{attribute addProperty BoxType "EK1122-0000-0018"}
{attribute addProperty Id "Beckhoff_EP2xxxsub_EK1100EK1100_179A0949162A_0001_EP2001_1000_0016EP2001_1F1194F38110.125A_0002_EP2001_1000_0017EP2001_1F1194F38110.125A_0003_EP2001_1000_0018EP2001_1F1194F38110.125A_0004_EP2001_1000_0019EP2001_1F1194F38110.125A_0005_EP2008_0001_0016EP2008_A854BE6D8110.125A_0006_EP2008_0001_0017EP2008_A854BE6D8110.125A_0007_EP2008_0001_0018EP2008_A854BE6D8110.125A_0008_EP2008_0001_0019EP2008_A854BE6D8110.125A_0009_EP2008_0002_0016EP2008_A854BE6D8110.125A_0010_EP2008_0002_0017EP2008_A854BE6D8110.125A_0011_EP2008_0002_0018EP2008_A854BE6D8110.125A_0012_EP2008_0002_0019EP2008_A854BE6D8110.125A_0013_EP2008_0022_0016EP2008_A854BE6D8110.125A_0014_EP2008_0022_0017EP2008_A854BE6D8110.125A_0015_EP2008_0022_0018EP2008_A854BE6D8110.125A_0016_EP2028_0001_0016EP2028_A854BE6D8110.125A_0017_EP2028_0001_0017EP2028_A854BE6D8110.125A_0018_EP2028_0001_0018EP2028_A854BE6D8110.125A_0019_EP2028_0002_0016EP2028_A854BE6D8110.125A_0020_EP2028_0002_0017EP2028_A854BE6D8110.125A_0021_EP2028_0002_0018EP2028_A854BE6D8110.125A_0022_EP2028_0002_0019EP2028_A854BE6D8110.125A_0023_EP2028_0032_0017EP2028_A854BE6D8110.125A_0024_EP2028_0032_0018EP2028_A854BE6D8110.125A_0025_EP2028_0032_0019EP2028_A854BE6D8110.125A_0026_EP2038_0001_0016EP2038_9444C9D314618.25A_0027_EP2038_0001_0017EP2038_9444C9D314618.25A_0028_EP2038_0001_0018EP2038_9444C9D314618.25A_0029_EP2038_0002_0016EP2038_9444C9D314618.25A_0030_EP2038_0002_0017EP2038_9444C9D314618.25A_0031_EP2038_0002_0018EP2038_9444C9D314618.25A_0032_EP2308_0000_0016EP2308_97B4DD118210.25A_0033_EP2308_0000_0017EP2308_97B4DD118210.25A_0034_EP2308_0000_0018EP2308_97B4DD118210.25A_0035_EP2308_0001_0016EP2308_97B4DD118210.25A_0036_EP2308_0001_0017EP2308_97B4DD118210.25A_0037_EP2308_0001_0018EP2308_97B4DD118210.25A_0038_EP2308_0001_0019EP2308_97B4DD118210.25A_0039_EP2308_0002_0016EP2308_97B4DD118210.25A_0040_EP2308_0002_0017EP2308_97B4DD118210.25A_0041_EP2308_0002_0018EP2308_97B4DD118210.25A_0042_EP2308_0002_0019EP2308_97B4DD118210.25A_0043_EP2316_0003_0016EP2316_7CBF98C533842.25A_0044_EP2316_0003_0017EP2316_7CBF98C533842.25A_0045_EP2316_0003_0018EP2316_7CBF98C533842.25A_0046_EP2316_0008_0016EP2316_9E547A1933041.25A_0047_EP2316_0008_0017EP2316_C551FFE833842.25A_0048_EP2316_0008_0018EP2316_4C10EA7633842.25A_0049_EP2316_0008_0019EP2316_7CBF98C533842.25A_0050_EP2316_0008_0020EP2316_7CBF98C533842.25A_0051_EP2316_0008_0021EP2316_7CBF98C533842.25A_0052_EP2318_0001_0016EP2318_97B4DD118210.25A_0053_EP2318_0001_0017EP2318_97B4DD118210.25A_0054_EP2318_0001_0018EP2318_97B4DD118210.25A_0055_EP2318_0001_0019EP2318_97B4DD118210.25A_0056_EP2318_0002_0016EP2318_97B4DD118210.25A_0057_EP2318_0002_0017EP2318_97B4DD118210.25A_0058_EP2318_0002_0018EP2318_97B4DD118210.25A_0059_EP2318_0002_0019EP2318_97B4DD118210.25A_0060_EP2328_0001_0016EP2328_97B4DD118210.25A_0061_EP2328_0001_0017EP2328_97B4DD118210.25A_0062_EP2328_0001_0018EP2328_97B4DD118210.25A_0063_EP2328_0002_0016EP2328_97B4DD118210.25A_0064_EP2328_0002_0017EP2328_97B4DD118210.25A_0065_EP2328_0002_0018EP2328_97B4DD118210.25A_0066_EP2328_0002_0019EP2328_97B4DD118210.25A_0067_EP2328_1061_0016EP2328_FBC9733E8210.25A_0068_EP2338_0001_0016EP2338_F9A026BF14618.25A_0069_EP2338_0001_0017EP2338_F9A026BF14618.25A_0070_EP2338_0001_0018EP2338_538B459D14618.25A_0071_EP2338_0001_0019EP2338_538B459D14618.25A_0072_EP2338_0001_0020EP2338_538B459D14618.25A_0073_EP2338_0001_0021EP2338_538B459D14618.25A_0074_EP2338_0001_0022EP2338_538B459D14618.25A_0075_EP2338_0001_0023EP2338_538B459D14618.25A_0076_EP2338_0002_0016EP2338_F9A026BF14618.25A_0077_EP2338_0002_0017EP2338_F9A026BF14618.25A_0078_EP2338_0002_0018EP2338_538B459D14618.25A_0079_EP2338_0002_0019EP2338_538B459D14618.25A_0080_EP2338_0002_0020EP2338_538B459D14618.25A_0081_EP2338_0002_0021EP2338_538B459D14618.25A_0082_EP2338_0002_0022EP2338_538B459D14618.25A_0083_EP2338_0002_0023EP2338_538B459D14618.25A_0084_EP2338_1001_0016EP2338_538B459D14618.25A_0085_EP2338_1001_0017EP2338_538B459D14618.25A_0086_EP2338_1001_0018EP2338_538B459D14618.25A_0087_EP2338_1002_0016EP2338_538B459D14618.25A_0088_EP2338_1002_0017EP2338_538B459D14618.25A_0089_EP2338_1002_0018EP2338_538B459D14618.25A_0090_EP2339_0003_0016EP2339_41D05C2438648.25A_0092_EP2339_0021_0016EP2339_FC6D243732240.25A_0093_EP2339_0021_0017EP2339_BBE0865932240.25A_0094_EP2339_0021_0018EP2339_BBE0865932240.25A_0095_EP2339_0021_0019EP2339_9219B49827434.25A_0096_EP2339_0021_0020EP2339_9219B49827434.25A_0097_EP2339_0022_0016EP2339_D59416F627434.25A_0098_EP2339_0022_0017EP2339_9219B49827434.25A_0099_EP2339_0022_0018EP2339_9219B49827434.25A_0100_EP2339_0022_0019EP2339_9219B49827434.25A_0101_EP2339_0042_0017EP2339_F4D25F8A8234359738378.25A_0102_EP2339_0042_0018EP2339_90CE4E13429496718668719476722.25A_0103_EP2339_0121_0016EP2339_9219B49827434.25A_0104_EP2349_0021_0016EP2349_9219B49827434.25A_0105_EP2349_0021_0017EP2349_9219B49827434.25A_0106_EP2349_0021_0018EP2349_9219B49827434.25A_0107_EP2349_0022_0016EP2349_9219B49827434.25A_0108_EP2349_0022_0017EP2349_9219B49827434.25A_0109_EP2349_0022_0018EP2349_9219B49827434.25A_0110_EP2624_0002_0016EP2624_4E3C7537496.125A_0111_EP2624_0002_0017EP2624_4E3C7537496.125A_0112_EP2624_0002_0018EP2624_4E3C7537496.125A_0113_EP2624_0002_0019EP2624_4E3C7537496.125A_0114_EP2809_0021_0016EP2809_859F43D214518.125A_0115_EP2809_0021_0017EP2809_859F43D214518.125A_0116_EP2809_0021_0018EP2809_859F43D214518.125A_0117_EP2809_0022_0016EP2809_859F43D214518.125A_0118_EP2809_0022_0017EP2809_859F43D214518.125A_0119_EP2809_0022_0018EP2809_859F43D214518.125A_0120_EP2809_0042_0017EP2809_15BF513E429496724934359738362.125A_0121_EP2809_0042_0018EP2809_556C4F60429496724934359738362.125A_0122_EP2816_0003_0016EP2816_E74B64DB39449.25A_0123_EP2816_0004_0016EP2816_68098FB020926.125A_0124_EP2816_0004_0017EP2816_E74B64DB39449.25A_0125_EP2816_0004_0018EP2816_E74B64DB39449.25A_0126_EP2816_0008_0016EP2816_18670F0939449.25A_0127_EP2816_0008_0017EP2816_18670F0939449.25A_0128_EP2816_0008_0018EP2816_5EA583C239449.25A_0129_EP2816_0008_0019EP2816_907EDA0F39449.25A_0130_EP2816_0008_0020EP2816_907EDA0F39449.25A_0131_EP2816_0008_0021EP2816_907EDA0F39449.25A_0132_EP2816_0010_0016EP2816_18670F0939449.25A_0133_EP2816_0010_0017EP2816_18670F0939449.25A_0134_EP2816_0010_0018EP2816_5EA583C239449.25A_0135_EP2816_0010_0019EP2816_907EDA0F39449.25A_0136_EP2816_0010_0020EP2816_907EDA0F39449.25A_0137_EP2816_0010_0021EP2816_907EDA0F39449.25A_0138_EP2817_0008_0016EP2817_AE3316D954668.25A_0139_EP2817_0008_0017EP2817_AE3316D954668.25A_0140_EP2817_0008_0018EP2817_AE3316D954668.25A_0141_EP2817_0008_0019EP2817_AE3316D954668.25"}
{attribute addProperty CRC "3477339297"}
{attribute addProperty SizeInBites "25538"}
{attribute addProperty SizeInBytes "171798695032.25"}
TYPE Beckhoff_EP2xxxEK1122_CF43FCA1 EXTENDS EK1122_179A0949 :
STRUCT
	{attribute addProperty Name "Beckhoff_EP2xxxsub_EK1100"}
	Beckhoff_EP2xxxsub_EK1100 : EK1100_179A0949;
	{attribute addProperty Name "A_0001_EP2001_1000_0016"}
	A_0001_EP2001_1000_0016 : EP2001_1F1194F3;
	{attribute addProperty Name "A_0002_EP2001_1000_0017"}
	A_0002_EP2001_1000_0017 : EP2001_1F1194F3;
	{attribute addProperty Name "A_0003_EP2001_1000_0018"}
	A_0003_EP2001_1000_0018 : EP2001_1F1194F3;
	{attribute addProperty Name "A_0004_EP2001_1000_0019"}
	A_0004_EP2001_1000_0019 : EP2001_1F1194F3;
	{attribute addProperty Name "A_0005_EP2008_0001_0016"}
	A_0005_EP2008_0001_0016 : EP2008_A854BE6D;
	{attribute addProperty Name "A_0006_EP2008_0001_0017"}
	A_0006_EP2008_0001_0017 : EP2008_A854BE6D;
	{attribute addProperty Name "A_0007_EP2008_0001_0018"}
	A_0007_EP2008_0001_0018 : EP2008_A854BE6D;
	{attribute addProperty Name "A_0008_EP2008_0001_0019"}
	A_0008_EP2008_0001_0019 : EP2008_A854BE6D;
	{attribute addProperty Name "A_0009_EP2008_0002_0016"}
	A_0009_EP2008_0002_0016 : EP2008_A854BE6D;
	{attribute addProperty Name "A_0010_EP2008_0002_0017"}
	A_0010_EP2008_0002_0017 : EP2008_A854BE6D;
	{attribute addProperty Name "A_0011_EP2008_0002_0018"}
	A_0011_EP2008_0002_0018 : EP2008_A854BE6D;
	{attribute addProperty Name "A_0012_EP2008_0002_0019"}
	A_0012_EP2008_0002_0019 : EP2008_A854BE6D;
	{attribute addProperty Name "A_0013_EP2008_0022_0016"}
	A_0013_EP2008_0022_0016 : EP2008_A854BE6D;
	{attribute addProperty Name "A_0014_EP2008_0022_0017"}
	A_0014_EP2008_0022_0017 : EP2008_A854BE6D;
	{attribute addProperty Name "A_0015_EP2008_0022_0018"}
	A_0015_EP2008_0022_0018 : EP2008_A854BE6D;
	{attribute addProperty Name "A_0016_EP2028_0001_0016"}
	A_0016_EP2028_0001_0016 : EP2028_A854BE6D;
	{attribute addProperty Name "A_0017_EP2028_0001_0017"}
	A_0017_EP2028_0001_0017 : EP2028_A854BE6D;
	{attribute addProperty Name "A_0018_EP2028_0001_0018"}
	A_0018_EP2028_0001_0018 : EP2028_A854BE6D;
	{attribute addProperty Name "A_0019_EP2028_0002_0016"}
	A_0019_EP2028_0002_0016 : EP2028_A854BE6D;
	{attribute addProperty Name "A_0020_EP2028_0002_0017"}
	A_0020_EP2028_0002_0017 : EP2028_A854BE6D;
	{attribute addProperty Name "A_0021_EP2028_0002_0018"}
	A_0021_EP2028_0002_0018 : EP2028_A854BE6D;
	{attribute addProperty Name "A_0022_EP2028_0002_0019"}
	A_0022_EP2028_0002_0019 : EP2028_A854BE6D;
	{attribute addProperty Name "A_0023_EP2028_0032_0017"}
	A_0023_EP2028_0032_0017 : EP2028_A854BE6D;
	{attribute addProperty Name "A_0024_EP2028_0032_0018"}
	A_0024_EP2028_0032_0018 : EP2028_A854BE6D;
	{attribute addProperty Name "A_0025_EP2028_0032_0019"}
	A_0025_EP2028_0032_0019 : EP2028_A854BE6D;
	{attribute addProperty Name "A_0026_EP2038_0001_0016"}
	A_0026_EP2038_0001_0016 : EP2038_9444C9D3;
	{attribute addProperty Name "A_0027_EP2038_0001_0017"}
	A_0027_EP2038_0001_0017 : EP2038_9444C9D3;
	{attribute addProperty Name "A_0028_EP2038_0001_0018"}
	A_0028_EP2038_0001_0018 : EP2038_9444C9D3;
	{attribute addProperty Name "A_0029_EP2038_0002_0016"}
	A_0029_EP2038_0002_0016 : EP2038_9444C9D3;
	{attribute addProperty Name "A_0030_EP2038_0002_0017"}
	A_0030_EP2038_0002_0017 : EP2038_9444C9D3;
	{attribute addProperty Name "A_0031_EP2038_0002_0018"}
	A_0031_EP2038_0002_0018 : EP2038_9444C9D3;
	{attribute addProperty Name "A_0032_EP2308_0000_0016"}
	A_0032_EP2308_0000_0016 : EP2308_97B4DD11;
	{attribute addProperty Name "A_0033_EP2308_0000_0017"}
	A_0033_EP2308_0000_0017 : EP2308_97B4DD11;
	{attribute addProperty Name "A_0034_EP2308_0000_0018"}
	A_0034_EP2308_0000_0018 : EP2308_97B4DD11;
	{attribute addProperty Name "A_0035_EP2308_0001_0016"}
	A_0035_EP2308_0001_0016 : EP2308_97B4DD11;
	{attribute addProperty Name "A_0036_EP2308_0001_0017"}
	A_0036_EP2308_0001_0017 : EP2308_97B4DD11;
	{attribute addProperty Name "A_0037_EP2308_0001_0018"}
	A_0037_EP2308_0001_0018 : EP2308_97B4DD11;
	{attribute addProperty Name "A_0038_EP2308_0001_0019"}
	A_0038_EP2308_0001_0019 : EP2308_97B4DD11;
	{attribute addProperty Name "A_0039_EP2308_0002_0016"}
	A_0039_EP2308_0002_0016 : EP2308_97B4DD11;
	{attribute addProperty Name "A_0040_EP2308_0002_0017"}
	A_0040_EP2308_0002_0017 : EP2308_97B4DD11;
	{attribute addProperty Name "A_0041_EP2308_0002_0018"}
	A_0041_EP2308_0002_0018 : EP2308_97B4DD11;
	{attribute addProperty Name "A_0042_EP2308_0002_0019"}
	A_0042_EP2308_0002_0019 : EP2308_97B4DD11;
	{attribute addProperty Name "A_0043_EP2316_0003_0016"}
	A_0043_EP2316_0003_0016 : EP2316_7CBF98C5;
	{attribute addProperty Name "A_0044_EP2316_0003_0017"}
	A_0044_EP2316_0003_0017 : EP2316_7CBF98C5;
	{attribute addProperty Name "A_0045_EP2316_0003_0018"}
	A_0045_EP2316_0003_0018 : EP2316_7CBF98C5;
	{attribute addProperty Name "A_0046_EP2316_0008_0016"}
	A_0046_EP2316_0008_0016 : EP2316_9E547A19;
	{attribute addProperty Name "A_0047_EP2316_0008_0017"}
	A_0047_EP2316_0008_0017 : EP2316_C551FFE8;
	{attribute addProperty Name "A_0048_EP2316_0008_0018"}
	A_0048_EP2316_0008_0018 : EP2316_4C10EA76;
	{attribute addProperty Name "A_0049_EP2316_0008_0019"}
	A_0049_EP2316_0008_0019 : EP2316_7CBF98C5;
	{attribute addProperty Name "A_0050_EP2316_0008_0020"}
	A_0050_EP2316_0008_0020 : EP2316_7CBF98C5;
	{attribute addProperty Name "A_0051_EP2316_0008_0021"}
	A_0051_EP2316_0008_0021 : EP2316_7CBF98C5;
	{attribute addProperty Name "A_0052_EP2318_0001_0016"}
	A_0052_EP2318_0001_0016 : EP2318_97B4DD11;
	{attribute addProperty Name "A_0053_EP2318_0001_0017"}
	A_0053_EP2318_0001_0017 : EP2318_97B4DD11;
	{attribute addProperty Name "A_0054_EP2318_0001_0018"}
	A_0054_EP2318_0001_0018 : EP2318_97B4DD11;
	{attribute addProperty Name "A_0055_EP2318_0001_0019"}
	A_0055_EP2318_0001_0019 : EP2318_97B4DD11;
	{attribute addProperty Name "A_0056_EP2318_0002_0016"}
	A_0056_EP2318_0002_0016 : EP2318_97B4DD11;
	{attribute addProperty Name "A_0057_EP2318_0002_0017"}
	A_0057_EP2318_0002_0017 : EP2318_97B4DD11;
	{attribute addProperty Name "A_0058_EP2318_0002_0018"}
	A_0058_EP2318_0002_0018 : EP2318_97B4DD11;
	{attribute addProperty Name "A_0059_EP2318_0002_0019"}
	A_0059_EP2318_0002_0019 : EP2318_97B4DD11;
	{attribute addProperty Name "A_0060_EP2328_0001_0016"}
	A_0060_EP2328_0001_0016 : EP2328_97B4DD11;
	{attribute addProperty Name "A_0061_EP2328_0001_0017"}
	A_0061_EP2328_0001_0017 : EP2328_97B4DD11;
	{attribute addProperty Name "A_0062_EP2328_0001_0018"}
	A_0062_EP2328_0001_0018 : EP2328_97B4DD11;
	{attribute addProperty Name "A_0063_EP2328_0002_0016"}
	A_0063_EP2328_0002_0016 : EP2328_97B4DD11;
	{attribute addProperty Name "A_0064_EP2328_0002_0017"}
	A_0064_EP2328_0002_0017 : EP2328_97B4DD11;
	{attribute addProperty Name "A_0065_EP2328_0002_0018"}
	A_0065_EP2328_0002_0018 : EP2328_97B4DD11;
	{attribute addProperty Name "A_0066_EP2328_0002_0019"}
	A_0066_EP2328_0002_0019 : EP2328_97B4DD11;
	{attribute addProperty Name "A_0067_EP2328_1061_0016"}
	A_0067_EP2328_1061_0016 : EP2328_FBC9733E;
	{attribute addProperty Name "A_0068_EP2338_0001_0016"}
	A_0068_EP2338_0001_0016 : EP2338_F9A026BF;
	{attribute addProperty Name "A_0069_EP2338_0001_0017"}
	A_0069_EP2338_0001_0017 : EP2338_F9A026BF;
	{attribute addProperty Name "A_0070_EP2338_0001_0018"}
	A_0070_EP2338_0001_0018 : EP2338_538B459D;
	{attribute addProperty Name "A_0071_EP2338_0001_0019"}
	A_0071_EP2338_0001_0019 : EP2338_538B459D;
	{attribute addProperty Name "A_0072_EP2338_0001_0020"}
	A_0072_EP2338_0001_0020 : EP2338_538B459D;
	{attribute addProperty Name "A_0073_EP2338_0001_0021"}
	A_0073_EP2338_0001_0021 : EP2338_538B459D;
	{attribute addProperty Name "A_0074_EP2338_0001_0022"}
	A_0074_EP2338_0001_0022 : EP2338_538B459D;
	{attribute addProperty Name "A_0075_EP2338_0001_0023"}
	A_0075_EP2338_0001_0023 : EP2338_538B459D;
	{attribute addProperty Name "A_0076_EP2338_0002_0016"}
	A_0076_EP2338_0002_0016 : EP2338_F9A026BF;
	{attribute addProperty Name "A_0077_EP2338_0002_0017"}
	A_0077_EP2338_0002_0017 : EP2338_F9A026BF;
	{attribute addProperty Name "A_0078_EP2338_0002_0018"}
	A_0078_EP2338_0002_0018 : EP2338_538B459D;
	{attribute addProperty Name "A_0079_EP2338_0002_0019"}
	A_0079_EP2338_0002_0019 : EP2338_538B459D;
	{attribute addProperty Name "A_0080_EP2338_0002_0020"}
	A_0080_EP2338_0002_0020 : EP2338_538B459D;
	{attribute addProperty Name "A_0081_EP2338_0002_0021"}
	A_0081_EP2338_0002_0021 : EP2338_538B459D;
	{attribute addProperty Name "A_0082_EP2338_0002_0022"}
	A_0082_EP2338_0002_0022 : EP2338_538B459D;
	{attribute addProperty Name "A_0083_EP2338_0002_0023"}
	A_0083_EP2338_0002_0023 : EP2338_538B459D;
	{attribute addProperty Name "A_0084_EP2338_1001_0016"}
	A_0084_EP2338_1001_0016 : EP2338_538B459D;
	{attribute addProperty Name "A_0085_EP2338_1001_0017"}
	A_0085_EP2338_1001_0017 : EP2338_538B459D;
	{attribute addProperty Name "A_0086_EP2338_1001_0018"}
	A_0086_EP2338_1001_0018 : EP2338_538B459D;
	{attribute addProperty Name "A_0087_EP2338_1002_0016"}
	A_0087_EP2338_1002_0016 : EP2338_538B459D;
	{attribute addProperty Name "A_0088_EP2338_1002_0017"}
	A_0088_EP2338_1002_0017 : EP2338_538B459D;
	{attribute addProperty Name "A_0089_EP2338_1002_0018"}
	A_0089_EP2338_1002_0018 : EP2338_538B459D;
	{attribute addProperty Name "A_0090_EP2339_0003_0016"}
	A_0090_EP2339_0003_0016 : EP2339_41D05C24;
	{attribute addProperty Name "A_0092_EP2339_0021_0016"}
	A_0092_EP2339_0021_0016 : EP2339_FC6D2437;
	{attribute addProperty Name "A_0093_EP2339_0021_0017"}
	A_0093_EP2339_0021_0017 : EP2339_BBE08659;
	{attribute addProperty Name "A_0094_EP2339_0021_0018"}
	A_0094_EP2339_0021_0018 : EP2339_BBE08659;
	{attribute addProperty Name "A_0095_EP2339_0021_0019"}
	A_0095_EP2339_0021_0019 : EP2339_9219B498;
	{attribute addProperty Name "A_0096_EP2339_0021_0020"}
	A_0096_EP2339_0021_0020 : EP2339_9219B498;
	{attribute addProperty Name "A_0097_EP2339_0022_0016"}
	A_0097_EP2339_0022_0016 : EP2339_D59416F6;
	{attribute addProperty Name "A_0098_EP2339_0022_0017"}
	A_0098_EP2339_0022_0017 : EP2339_9219B498;
	{attribute addProperty Name "A_0099_EP2339_0022_0018"}
	A_0099_EP2339_0022_0018 : EP2339_9219B498;
	{attribute addProperty Name "A_0100_EP2339_0022_0019"}
	A_0100_EP2339_0022_0019 : EP2339_9219B498;
	{attribute addProperty Name "A_0101_EP2339_0042_0017"}
	A_0101_EP2339_0042_0017 : EP2339_F4D25F8A;
	{attribute addProperty Name "A_0102_EP2339_0042_0018"}
	A_0102_EP2339_0042_0018 : EP2339_90CE4E13;
	{attribute addProperty Name "A_0103_EP2339_0121_0016"}
	A_0103_EP2339_0121_0016 : EP2339_9219B498;
	{attribute addProperty Name "A_0104_EP2349_0021_0016"}
	A_0104_EP2349_0021_0016 : EP2349_9219B498;
	{attribute addProperty Name "A_0105_EP2349_0021_0017"}
	A_0105_EP2349_0021_0017 : EP2349_9219B498;
	{attribute addProperty Name "A_0106_EP2349_0021_0018"}
	A_0106_EP2349_0021_0018 : EP2349_9219B498;
	{attribute addProperty Name "A_0107_EP2349_0022_0016"}
	A_0107_EP2349_0022_0016 : EP2349_9219B498;
	{attribute addProperty Name "A_0108_EP2349_0022_0017"}
	A_0108_EP2349_0022_0017 : EP2349_9219B498;
	{attribute addProperty Name "A_0109_EP2349_0022_0018"}
	A_0109_EP2349_0022_0018 : EP2349_9219B498;
	{attribute addProperty Name "A_0110_EP2624_0002_0016"}
	A_0110_EP2624_0002_0016 : EP2624_4E3C7537;
	{attribute addProperty Name "A_0111_EP2624_0002_0017"}
	A_0111_EP2624_0002_0017 : EP2624_4E3C7537;
	{attribute addProperty Name "A_0112_EP2624_0002_0018"}
	A_0112_EP2624_0002_0018 : EP2624_4E3C7537;
	{attribute addProperty Name "A_0113_EP2624_0002_0019"}
	A_0113_EP2624_0002_0019 : EP2624_4E3C7537;
	{attribute addProperty Name "A_0114_EP2809_0021_0016"}
	A_0114_EP2809_0021_0016 : EP2809_859F43D2;
	{attribute addProperty Name "A_0115_EP2809_0021_0017"}
	A_0115_EP2809_0021_0017 : EP2809_859F43D2;
	{attribute addProperty Name "A_0116_EP2809_0021_0018"}
	A_0116_EP2809_0021_0018 : EP2809_859F43D2;
	{attribute addProperty Name "A_0117_EP2809_0022_0016"}
	A_0117_EP2809_0022_0016 : EP2809_859F43D2;
	{attribute addProperty Name "A_0118_EP2809_0022_0017"}
	A_0118_EP2809_0022_0017 : EP2809_859F43D2;
	{attribute addProperty Name "A_0119_EP2809_0022_0018"}
	A_0119_EP2809_0022_0018 : EP2809_859F43D2;
	{attribute addProperty Name "A_0120_EP2809_0042_0017"}
	A_0120_EP2809_0042_0017 : EP2809_15BF513E;
	{attribute addProperty Name "A_0121_EP2809_0042_0018"}
	A_0121_EP2809_0042_0018 : EP2809_556C4F60;
	{attribute addProperty Name "A_0122_EP2816_0003_0016"}
	A_0122_EP2816_0003_0016 : EP2816_E74B64DB;
	{attribute addProperty Name "A_0123_EP2816_0004_0016"}
	A_0123_EP2816_0004_0016 : EP2816_68098FB0;
	{attribute addProperty Name "A_0124_EP2816_0004_0017"}
	A_0124_EP2816_0004_0017 : EP2816_E74B64DB;
	{attribute addProperty Name "A_0125_EP2816_0004_0018"}
	A_0125_EP2816_0004_0018 : EP2816_E74B64DB;
	{attribute addProperty Name "A_0126_EP2816_0008_0016"}
	A_0126_EP2816_0008_0016 : EP2816_18670F09;
	{attribute addProperty Name "A_0127_EP2816_0008_0017"}
	A_0127_EP2816_0008_0017 : EP2816_18670F09;
	{attribute addProperty Name "A_0128_EP2816_0008_0018"}
	A_0128_EP2816_0008_0018 : EP2816_5EA583C2;
	{attribute addProperty Name "A_0129_EP2816_0008_0019"}
	A_0129_EP2816_0008_0019 : EP2816_907EDA0F;
	{attribute addProperty Name "A_0130_EP2816_0008_0020"}
	A_0130_EP2816_0008_0020 : EP2816_907EDA0F;
	{attribute addProperty Name "A_0131_EP2816_0008_0021"}
	A_0131_EP2816_0008_0021 : EP2816_907EDA0F;
	{attribute addProperty Name "A_0132_EP2816_0010_0016"}
	A_0132_EP2816_0010_0016 : EP2816_18670F09;
	{attribute addProperty Name "A_0133_EP2816_0010_0017"}
	A_0133_EP2816_0010_0017 : EP2816_18670F09;
	{attribute addProperty Name "A_0134_EP2816_0010_0018"}
	A_0134_EP2816_0010_0018 : EP2816_5EA583C2;
	{attribute addProperty Name "A_0135_EP2816_0010_0019"}
	A_0135_EP2816_0010_0019 : EP2816_907EDA0F;
	{attribute addProperty Name "A_0136_EP2816_0010_0020"}
	A_0136_EP2816_0010_0020 : EP2816_907EDA0F;
	{attribute addProperty Name "A_0137_EP2816_0010_0021"}
	A_0137_EP2816_0010_0021 : EP2816_907EDA0F;
	{attribute addProperty Name "A_0138_EP2817_0008_0016"}
	A_0138_EP2817_0008_0016 : EP2817_AE3316D9;
	{attribute addProperty Name "A_0139_EP2817_0008_0017"}
	A_0139_EP2817_0008_0017 : EP2817_AE3316D9;
	{attribute addProperty Name "A_0140_EP2817_0008_0018"}
	A_0140_EP2817_0008_0018 : EP2817_AE3316D9;
	{attribute addProperty Name "A_0141_EP2817_0008_0019"}
	A_0141_EP2817_0008_0019 : EP2817_AE3316D9;
END_STRUCT
END_TYPE

(* stored: Version 1.2.0.0, ProductVersion 3.1.4024.9
   DUT Beckhoff_EP2xxxEK1122_CF43FCA1: Id {097468ee-0c25-4230-80a4-031dfc389b1b} *)
